(* IEC 61131-3 sources: AXOpen/src/components.dukane.welders/ctrl/src/TemplateComponent (part 2) *)

                IF Config.HWIDs.HwID_out_1  = UINT#0 THEN
                    Messenger.Activate(UINT#1152,eAxoMessageCategory#Error);
                    Status.Error.Id := UINT#1152;
                    RETURN;
                END_IF;
                IF Config.HWIDs.HwID_out_2  = UINT#0 THEN
                    Messenger.Activate(UINT#1153,eAxoMessageCategory#Error);
                    Status.Error.Id := UINT#1153;
                    RETURN;
                END_IF;
                IF Config.HWIDs.HwID_out_3  = UINT#0 THEN
                    Messenger.Activate(UINT#1154,eAxoMessageCategory#Error);
                    Status.Error.Id := UINT#1154;
                    RETURN;
                END_IF;
                IF Config.HWIDs.HwID_out_4  = UINT#0 THEN
                    Messenger.Activate(UINT#1155,eAxoMessageCategory#Error);
                    Status.Error.Id := UINT#1155;
                    RETURN;
                END_IF;
                IF Config.HWIDs.HwID_out_5  = UINT#0 THEN
                    Messenger.Activate(UINT#1156,eAxoMessageCategory#Error);
                    Status.Error.Id := UINT#1156;
                    RETURN;
                END_IF;
                IF Config.HWIDs.HwID_out_6  = UINT#0 THEN
                    Messenger.Activate(UINT#1157,eAxoMessageCategory#Error);
                    Status.Error.Id := UINT#1157;
                    RETURN;
                END_IF;
                IF Config.HWIDs.HwID_out_7  = UINT#0 THEN
                    Messenger.Activate(UINT#1158,eAxoMessageCategory#Error);
                    Status.Error.Id := UINT#1158;
                    RETURN;
                END_IF;
                IF Config.HWIDs.HwID_out_8  = UINT#0 THEN
                    Messenger.Activate(UINT#1159,eAxoMessageCategory#Error);
                    Status.Error.Id := UINT#1159;
                    RETURN;
                END_IF;
                IF Config.HWIDs.HwID_out_9  = UINT#0 THEN
                    Messenger.Activate(UINT#1160,eAxoMessageCategory#Error);
                    Status.Error.Id := UINT#1160;
                    RETURN;
                END_IF;
                IF Config.HWIDs.HwID_out_10  = UINT#0 THEN
                    Messenger.Activate(UINT#1161,eAxoMessageCategory#Error);
                    Status.Error.Id := UINT#1161;
                    RETURN;
                END_IF;
                IF Config.HWIDs.HwID_out_11  = UINT#0 THEN
                    Messenger.Activate(UINT#1162,eAxoMessageCategory#Error);
                    Status.Error.Id := UINT#1162;
                    RETURN;
                END_IF;
                IF Config.HWIDs.HwID_out_12  = UINT#0 THEN
                    Messenger.Activate(UINT#1163,eAxoMessageCategory#Error);
                    Status.Error.Id := UINT#1163;
                    RETURN;
                END_IF;
                IF Config.HWIDs.HwID_out_13  = UINT#0 THEN
                    Messenger.Activate(UINT#1164,eAxoMessageCategory#Error);
                    Status.Error.Id := UINT#1164;
                    RETURN;
                END_IF;
                IF Config.HWIDs.HwID_out_14  = UINT#0 THEN
                    Messenger.Activate(UINT#1165,eAxoMessageCategory#Error);
                    Status.Error.Id := UINT#1165;
                    RETURN;
                END_IF;
                IF Config.HWIDs.HwID_out_15  = UINT#0 THEN
                    Messenger.Activate(UINT#1166,eAxoMessageCategory#Error);
                    Status.Error.Id := UINT#1166;
                    RETURN;
                END_IF;
                IF Config.HWIDs.HwID_out_16  = UINT#0 THEN
                    Messenger.Activate(UINT#1167,eAxoMessageCategory#Error);
                    Status.Error.Id := UINT#1167;
                    RETURN;
                END_IF;
                IF Config.HWIDs.HwID_out_17  = UINT#0 THEN
                    Messenger.Activate(UINT#1168,eAxoMessageCategory#Error);
                    Status.Error.Id := UINT#1168;
                    RETURN;
                END_IF;
                IF Config.HWIDs.HwID_out_18  = UINT#0 THEN
                    Messenger.Activate(UINT#1169,eAxoMessageCategory#Error);
                    Status.Error.Id := UINT#1169;
                    RETURN;
                END_IF;
                IF Config.HWIDs.HwID_out_19  = UINT#0 THEN
                    Messenger.Activate(UINT#1170,eAxoMessageCategory#Error);
                    Status.Error.Id := UINT#1170;
                    RETURN;
                END_IF;
                IF Config.HWIDs.HwID_out_20  = UINT#0 THEN
                    Messenger.Activate(UINT#1171,eAxoMessageCategory#Error);
                    Status.Error.Id := UINT#1171;
                    RETURN;
                END_IF;

                _initHwCheckDone    := TRUE;
            END_IF;

            //***********Update inputs **************
            _retVal := Siemens.Simatic.S71500.DistributedIO.ReadData(TO_WORD(Config.HWIDs.HwID_in_1) ,_data_in);
            IF _retVal > WORD#0 THEN
                Messenger.Activate(UINT#1201, eAxoMessageCategory#ProgrammingError);
                Status.Error.Id := UINT#1201;
                RETURN;
            END_IF;

            // TemplateComponentInputStructure_hwID_in_1.Item1  :=      _data_in[0].%X0;
            // TemplateComponentInputStructure_hwID_in_1.Item2  :=      _data_in[0].%X1;
            // TemplateComponentInputStructure_hwID_in_1.Item3  :=      _data_in[0].%X2;
            // TemplateComponentInputStructure_hwID_in_1.Item4  :=      _data_in[0].%X3;
            // TemplateComponentInputStructure_hwID_in_1.Item5  :=      _data_in[0].%X4;

            _retVal := Siemens.Simatic.S71500.DistributedIO.ReadData(TO_WORD(Config.HWIDs.HwID_in_2) ,_data_in);
            IF _retVal > WORD#0 THEN
                Messenger.Activate(UINT#1202, eAxoMessageCategory#ProgrammingError);
                Status.Error.Id := UINT#1202;
                RETURN;
            END_IF;

            // TemplateComponentInputStructure_hwID_in_2.Item1  :=      _data_in[0].%X0;
            // TemplateComponentInputStructure_hwID_in_2.Item2  :=      _data_in[0].%X1;
            // TemplateComponentInputStructure_hwID_in_2.Item3  :=      _data_in[0].%X2;
            // TemplateComponentInputStructure_hwID_in_2.Item4  :=      _data_in[0].%X3;
            // TemplateComponentInputStructure_hwID_in_2.Item5  :=      _data_in[0].%X4;

            _retVal := Siemens.Simatic.S71500.DistributedIO.ReadData(TO_WORD(Config.HWIDs.HwID_in_3) ,_data_in);
            IF _retVal > WORD#0 THEN
                Messenger.Activate(UINT#1203, eAxoMessageCategory#ProgrammingError);
                Status.Error.Id := UINT#1203;
                RETURN;
            END_IF;

            // TemplateComponentInputStructure_hwID_in_3.Item1  :=      _data_in[0].%X0;
            // TemplateComponentInputStructure_hwID_in_3.Item2  :=      _data_in[0].%X1;
            // TemplateComponentInputStructure_hwID_in_3.Item3  :=      _data_in[0].%X2;
            // TemplateComponentInputStructure_hwID_in_3.Item4  :=      _data_in[0].%X3;
            // TemplateComponentInputStructure_hwID_in_3.Item5  :=      _data_in[0].%X4;

            _retVal := Siemens.Simatic.S71500.DistributedIO.ReadData(TO_WORD(Config.HWIDs.HwID_in_4) ,_data_in);
            IF _retVal > WORD#0 THEN
                Messenger.Activate(UINT#1204, eAxoMessageCategory#ProgrammingError);
                Status.Error.Id := UINT#1204;
                RETURN;
            END_IF;

            // TemplateComponentInputStructure_hwID_in_4.Item1  :=      _data_in[0].%X0;
            // TemplateComponentInputStructure_hwID_in_4.Item2  :=      _data_in[0].%X1;
            // TemplateComponentInputStructure_hwID_in_4.Item3  :=      _data_in[0].%X2;
            // TemplateComponentInputStructure_hwID_in_4.Item4  :=      _data_in[0].%X3;
            // TemplateComponentInputStructure_hwID_in_4.Item5  :=      _data_in[0].%X4;

            _retVal := Siemens.Simatic.S71500.DistributedIO.ReadData(TO_WORD(Config.HWIDs.HwID_in_5) ,_data_in);
            IF _retVal > WORD#0 THEN
                Messenger.Activate(UINT#1205, eAxoMessageCategory#ProgrammingError);
                Status.Error.Id := UINT#1205;
                RETURN;
            END_IF;

            // TemplateComponentInputStructure_hwID_in_5.Item1  :=      _data_in[0].%X0;
            // TemplateComponentInputStructure_hwID_in_5.Item2  :=      _data_in[0].%X1;
            // TemplateComponentInputStructure_hwID_in_5.Item3  :=      _data_in[0].%X2;
            // TemplateComponentInputStructure_hwID_in_5.Item4  :=      _data_in[0].%X3;
            // TemplateComponentInputStructure_hwID_in_5.Item5  :=      _data_in[0].%X4;

            _retVal := Siemens.Simatic.S71500.DistributedIO.ReadData(TO_WORD(Config.HWIDs.HwID_in_6) ,_data_in);
            IF _retVal > WORD#0 THEN
                Messenger.Activate(UINT#1206, eAxoMessageCategory#ProgrammingError);
                Status.Error.Id := UINT#1206;
                RETURN;
            END_IF;

            // _word.%B1                                                           :=  _data_in[0];
            // _word.%B0                                                           :=  _data_in[1];
            // TemplateComponentInputStructure_hwID_in_6.Item1                     :=  TO_UINT(_word);
            // _word.%B1                                                           :=  _data_in[2];
            // _word.%B0                                                           :=  _data_in[3];
            // TemplateComponentInputStructure_hwID_in_6.Item2                     :=  TO_UINT(_word);
            // _word.%B1                                                           :=  _data_in[4];
            // _word.%B0                                                           :=  _data_in[5];
            // TemplateComponentInputStructure_hwID_in_6.Item3                     :=  TO_UINT(_word);
            // _word.%B1                                                           :=  _data_in[6];
            // _word.%B0                                                           :=  _data_in[7];
            // TemplateComponentInputStructure_hwID_in_6.Item4                     :=  TO_UINT(_word);

            _retVal := Siemens.Simatic.S71500.DistributedIO.ReadData(TO_WORD(Config.HWIDs.HwID_in_7) ,_data_in);
            IF _retVal > WORD#0 THEN
                Messenger.Activate(UINT#1207, eAxoMessageCategory#ProgrammingError);
                Status.Error.Id := UINT#1207;
                RETURN;
            END_IF;

            // _dword.%B3                                                          :=  _data_in[0];
            // _dword.%B2                                                          :=  _data_in[1];
            // _dword.%B1                                                          :=  _data_in[2];
            // _dword.%B0                                                          :=  _data_in[3];
            // TemplateComponentInputStructure_hwID_in_7.Item1                     :=  TO_DINT(_dword);
            // _dword.%B3                                                          :=  _data_in[4];
            // _dword.%B2                                                          :=  _data_in[5];
            // _dword.%B1                                                          :=  _data_in[6];
            // _dword.%B0                                                          :=  _data_in[7];
            // TemplateComponentInputStructure_hwID_in_7.Item2                     :=  TO_REAL(_dword);

            _retVal := Siemens.Simatic.S71500.DistributedIO.ReadData(TO_WORD(Config.HWIDs.HwID_in_8) ,_data_in);
            IF _retVal > WORD#0 THEN
                Messenger.Activate(UINT#1208, eAxoMessageCategory#ProgrammingError);
                Status.Error.Id := UINT#1208;
                RETURN;
            END_IF;

            // _dword.%B3                                                          :=  _data_in[0];
            // _dword.%B2                                                          :=  _data_in[1];
            // _dword.%B1                                                          :=  _data_in[2];
            // _dword.%B0                                                          :=  _data_in[3];
            // TemplateComponentInputStructure_hwID_in_8.Item1                     :=  TO_DINT(_dword);
            // _dword.%B3                                                          :=  _data_in[4];
            // _dword.%B2                                                          :=  _data_in[5];
            // _dword.%B1                                                          :=  _data_in[6];
            // _dword.%B0                                                          :=  _data_in[7];
            // TemplateComponentInputStructure_hwID_in_8.Item2                     :=  TO_REAL(_dword);

            _retVal := Siemens.Simatic.S71500.DistributedIO.ReadData(TO_WORD(Config.HWIDs.HwID_in_9) ,_data_in);
            IF _retVal > WORD#0 THEN
                Messenger.Activate(UINT#1209, eAxoMessageCategory#ProgrammingError);
                Status.Error.Id := UINT#1209;
                RETURN;
            END_IF;

            // _dword.%B3                                                          :=  _data_in[0];
            // _dword.%B2                                                          :=  _data_in[1];
            // _dword.%B1                                                          :=  _data_in[2];
            // _dword.%B0                                                          :=  _data_in[3];
            // TemplateComponentInputStructure_hwID_in_9.Item1                     :=  TO_DINT(_dword);
            // _dword.%B3                                                          :=  _data_in[4];
            // _dword.%B2                                                          :=  _data_in[5];
            // _dword.%B1                                                          :=  _data_in[6];
            // _dword.%B0                                                          :=  _data_in[7];
            // TemplateComponentInputStructure_hwID_in_9.Item2                     :=  TO_REAL(_dword);

            _retVal := Siemens.Simatic.S71500.DistributedIO.ReadData(TO_WORD(Config.HWIDs.HwID_in_10) ,_data_in);
            IF _retVal > WORD#0 THEN
                Messenger.Activate(UINT#1210, eAxoMessageCategory#ProgrammingError);
                Status.Error.Id := UINT#1210;
                RETURN;
            END_IF;

            // _dword.%B3                                                          :=  _data_in[0];
            // _dword.%B2                                                          :=  _data_in[1];
            // _dword.%B1                                                          :=  _data_in[2];
            // _dword.%B0                                                          :=  _data_in[3];
            // TemplateComponentInputStructure_hwID_in_10.Item1                    :=  TO_DINT(_dword);
            // _dword.%B3                                                          :=  _data_in[4];
            // _dword.%B2                                                          :=  _data_in[5];
            // _dword.%B1                                                          :=  _data_in[6];
            // _dword.%B0                                                          :=  _data_in[7];
            // TemplateComponentInputStructure_hwID_in_10.Item2                    :=  TO_REAL(_dword);

            _retVal := Siemens.Simatic.S71500.DistributedIO.ReadData(TO_WORD(Config.HWIDs.HwID_in_11) ,_data_in);
            IF _retVal > WORD#0 THEN
                Messenger.Activate(UINT#1211, eAxoMessageCategory#ProgrammingError);
                Status.Error.Id := UINT#1211;
                RETURN;
            END_IF;

            // TemplateComponentInputStructure_hwID_in_11.Item1  :=      _data_in[0].%X0;
            // TemplateComponentInputStructure_hwID_in_11.Item2  :=      _data_in[0].%X1;
            // TemplateComponentInputStructure_hwID_in_11.Item3  :=      _data_in[0].%X2;
            // TemplateComponentInputStructure_hwID_in_11.Item4  :=      _data_in[0].%X3;
            // TemplateComponentInputStructure_hwID_in_11.Item5  :=      _data_in[0].%X4;

            _retVal := Siemens.Simatic.S71500.DistributedIO.ReadData(TO_WORD(Config.HWIDs.HwID_in_12) ,_data_in);
            IF _retVal > WORD#0 THEN
                Messenger.Activate(UINT#1212, eAxoMessageCategory#ProgrammingError);
                Status.Error.Id := UINT#1212;
                RETURN;
            END_IF;

            // TemplateComponentInputStructure_hwID_in_12.Item1  :=      _data_in[0].%X0;
            // TemplateComponentInputStructure_hwID_in_12.Item2  :=      _data_in[0].%X1;
            // TemplateComponentInputStructure_hwID_in_12.Item3  :=      _data_in[0].%X2;
            // TemplateComponentInputStructure_hwID_in_12.Item4  :=      _data_in[0].%X3;
            // TemplateComponentInputStructure_hwID_in_12.Item5  :=      _data_in[0].%X4;

            _retVal := Siemens.Simatic.S71500.DistributedIO.ReadData(TO_WORD(Config.HWIDs.HwID_in_13) ,_data_in);
            IF _retVal > WORD#0 THEN
                Messenger.Activate(UINT#1213, eAxoMessageCategory#ProgrammingError);
                Status.Error.Id := UINT#1213;
                RETURN;
            END_IF;

            // TemplateComponentInputStructure_hwID_in_13.Item1  :=      _data_in[0].%X0;
            // TemplateComponentInputStructure_hwID_in_13.Item2  :=      _data_in[0].%X1;
            // TemplateComponentInputStructure_hwID_in_13.Item3  :=      _data_in[0].%X2;
            // TemplateComponentInputStructure_hwID_in_13.Item4  :=      _data_in[0].%X3;
            // TemplateComponentInputStructure_hwID_in_13.Item5  :=      _data_in[0].%X4;

            _retVal := Siemens.Simatic.S71500.DistributedIO.ReadData(TO_WORD(Config.HWIDs.HwID_in_14) ,_data_in);
            IF _retVal > WORD#0 THEN
                Messenger.Activate(UINT#1214, eAxoMessageCategory#ProgrammingError);
                Status.Error.Id := UINT#1214;
                RETURN;
            END_IF;

            // TemplateComponentInputStructure_hwID_in_14.Item1  :=      _data_in[0].%X0;
            // TemplateComponentInputStructure_hwID_in_14.Item2  :=      _data_in[0].%X1;
            // TemplateComponentInputStructure_hwID_in_14.Item3  :=      _data_in[0].%X2;
            // TemplateComponentInputStructure_hwID_in_14.Item4  :=      _data_in[0].%X3;
            // TemplateComponentInputStructure_hwID_in_14.Item5  :=      _data_in[0].%X4;

            _retVal := Siemens.Simatic.S71500.DistributedIO.ReadData(TO_WORD(Config.HWIDs.HwID_in_15) ,_data_in);
            IF _retVal > WORD#0 THEN
                Messenger.Activate(UINT#1215, eAxoMessageCategory#ProgrammingError);
                Status.Error.Id := UINT#1215;
                RETURN;
            END_IF;

            // TemplateComponentInputStructure_hwID_in_15.Item1  :=      _data_in[0].%X0;
            // TemplateComponentInputStructure_hwID_in_15.Item2  :=      _data_in[0].%X1;
            // TemplateComponentInputStructure_hwID_in_15.Item3  :=      _data_in[0].%X2;
            // TemplateComponentInputStructure_hwID_in_15.Item4  :=      _data_in[0].%X3;
            // TemplateComponentInputStructure_hwID_in_15.Item5  :=      _data_in[0].%X4;

            _retVal := Siemens.Simatic.S71500.DistributedIO.ReadData(TO_WORD(Config.HWIDs.HwID_in_16) ,_data_in);
            IF _retVal > WORD#0 THEN
                Messenger.Activate(UINT#1216, eAxoMessageCategory#ProgrammingError);
                Status.Error.Id := UINT#1216;
                RETURN;
            END_IF;

            // _word.%B1                                                           :=  _data_in[0];
            // _word.%B0                                                           :=  _data_in[1];
            // TemplateComponentInputStructure_hwID_in_16.Item1                    :=  TO_UINT(_word);
            // _word.%B1                                                           :=  _data_in[2];
            // _word.%B0                                                           :=  _data_in[3];
            // TemplateComponentInputStructure_hwID_in_16.Item2                    :=  TO_UINT(_word);
            // _word.%B1                                                           :=  _data_in[4];
            // _word.%B0                                                           :=  _data_in[5];
            // TemplateComponentInputStructure_hwID_in_16.Item3                    :=  TO_UINT(_word);
            // _word.%B1                                                           :=  _data_in[6];
            // _word.%B0                                                           :=  _data_in[7];
            // TemplateComponentInputStructure_hwID_in_16.Item4                    :=  TO_UINT(_word);

            _retVal := Siemens.Simatic.S71500.DistributedIO.ReadData(TO_WORD(Config.HWIDs.HwID_in_17) ,_data_in);
            IF _retVal > WORD#0 THEN
                Messenger.Activate(UINT#1217, eAxoMessageCategory#ProgrammingError);
                Status.Error.Id := UINT#1217;
                RETURN;
            END_IF;

            // _dword.%B3                                                          :=  _data_in[0];
            // _dword.%B2                                                          :=  _data_in[1];
            // _dword.%B1                                                          :=  _data_in[2];
            // _dword.%B0                                                          :=  _data_in[3];
            // TemplateComponentInputStructure_hwID_in_17.Item1                    :=  TO_DINT(_dword);
            // _dword.%B3                                                          :=  _data_in[4];
            // _dword.%B2                                                          :=  _data_in[5];
            // _dword.%B1                                                          :=  _data_in[6];
            // _dword.%B0                                                          :=  _data_in[7];
            // TemplateComponentInputStructure_hwID_in_17.Item2                    :=  TO_REAL(_dword);

            _retVal := Siemens.Simatic.S71500.DistributedIO.ReadData(TO_WORD(Config.HWIDs.HwID_in_18) ,_data_in);
            IF _retVal > WORD#0 THEN
                Messenger.Activate(UINT#1218, eAxoMessageCategory#ProgrammingError);
                Status.Error.Id := UINT#1218;
                RETURN;
            END_IF;

            // _dword.%B3                                                          :=  _data_in[0];
            // _dword.%B2                                                          :=  _data_in[1];
            // _dword.%B1                                                          :=  _data_in[2];
            // _dword.%B0                                                          :=  _data_in[3];
            // TemplateComponentInputStructure_hwID_in_18.Item1                    :=  TO_DINT(_dword);
            // _dword.%B3                                                          :=  _data_in[4];
            // _dword.%B2                                                          :=  _data_in[5];
            // _dword.%B1                                                          :=  _data_in[6];
            // _dword.%B0                                                          :=  _data_in[7];
            // TemplateComponentInputStructure_hwID_in_18.Item2                    :=  TO_REAL(_dword);

            _retVal := Siemens.Simatic.S71500.DistributedIO.ReadData(TO_WORD(Config.HWIDs.HwID_in_19) ,_data_in);
            IF _retVal > WORD#0 THEN
                Messenger.Activate(UINT#1219, eAxoMessageCategory#ProgrammingError);
                Status.Error.Id := UINT#1219;
                RETURN;
            END_IF;

            // _dword.%B3                                                          :=  _data_in[0];
            // _dword.%B2                                                          :=  _data_in[1];
            // _dword.%B1                                                          :=  _data_in[2];
            // _dword.%B0                                                          :=  _data_in[3];
            // TemplateComponentInputStructure_hwID_in_19.Item1                    :=  TO_DINT(_dword);
            // _dword.%B3                                                          :=  _data_in[4];
            // _dword.%B2                                                          :=  _data_in[5];
            // _dword.%B1                                                          :=  _data_in[6];
            // _dword.%B0                                                          :=  _data_in[7];
            // TemplateComponentInputStructure_hwID_in_19.Item2                    :=  TO_REAL(_dword);

            _retVal := Siemens.Simatic.S71500.DistributedIO.ReadData(TO_WORD(Config.HWIDs.HwID_in_20) ,_data_in);
            IF _retVal > WORD#0 THEN
                Messenger.Activate(UINT#1220, eAxoMessageCategory#ProgrammingError);
                Status.Error.Id := UINT#1220;
                RETURN;
            END_IF;

            // _dword.%B3                                                          :=  _data_in[0];
            // _dword.%B2                                                          :=  _data_in[1];
            // _dword.%B1                                                          :=  _data_in[2];
            // _dword.%B0                                                          :=  _data_in[3];
            // TemplateComponentInputStructure_hwID_in_20.Item1                    :=  TO_DINT(_dword);
            // _dword.%B3                                                          :=  _data_in[4];
            // _dword.%B2                                                          :=  _data_in[5];
            // _dword.%B1                                                          :=  _data_in[6];
            // _dword.%B0                                                          :=  _data_in[7];
            // TemplateComponentInputStructure_hwID_in_20.Item2                    :=  TO_REAL(_dword);

            //*************INITIALIZATION*************
            RestoreTask.Run(THIS);
            TemplateTask_10steps_1.Run(THIS);
            TemplateTask_10steps_2.Run(THIS);
            TemplateTask_10steps_3.Run(THIS);
            TemplateTask_10steps_4.Run(THIS);
            TemplateTask_10steps_5.Run(THIS);
            TemplateTask_10steps_6.Run(THIS);
            TemplateTask_20steps_1.Run(THIS);
            TemplateTask_20steps_2.Run(THIS);
            TemplateTask_20steps_3.Run(THIS);
            TemplateTask_20steps_4.Run(THIS);
            TemplateTask_20steps_5.Run(THIS);
            TemplateTask_20steps_6.Run(THIS);

            //****************************************

            //********************Diagnostics*********
            HardwareDiagnosticsTask.Run(THIS,Config.HWIDs.HW_Device);
            //****************************************

            //*************RESTORE********************
            RestoreTask.SetIsDisabled(FALSE);
            IF RestoreTask.Execute(THIS) THEN
                THIS.Restore();
            END_IF;
            //****************************************

            //*************TemplateTask_10steps_1**************
            TemplateTask_10steps_1.SetIsDisabled(FALSE);
            IF TemplateTask_10steps_1.StartTriggered() THEN
                Status.Action.Id :=  UINT#100;
            END_IF;
            Messenger.ActivateOnCondition(ULINT#100,TemplateTask_10steps_1.IsBusy(), eAxoMessageCategory#Info);
            Messenger.ActivateOnCondition(ULINT#101,TemplateTask_10steps_1.IsDone(), eAxoMessageCategory#Info);
            IF TemplateTask_10steps_1.Execute(THIS) THEN
                IF _progress = 0 THEN
                    Status.Error.Id := UINT#0;
                    TaskMessenger.Restore();
                    THIS.CallTimers(FALSE);
                    _progress := 300;
                END_IF;

                IF _progress = 300 THEN                                                                                     // TemplateTask_10steps_1 running: , add_the_detailed_description_of_the_current_action_1
                    IF _infoTimer.output THEN
                        TaskMessenger.Activate( UINT#500, eAxoMessageCategory#Warning);
                        Status.Error.Id :=      UINT#500;
                    END_IF;

                    IF TRUE THEN
                        THIS.CallTimers(FALSE);
                        _progress := 301;
                    END_IF;
                END_IF;

                IF _progress = 301 THEN                                                                                     // TemplateTask_10steps_1 running: , add_the_detailed_description_of_the_current_action_2
                    IF _infoTimer.output THEN
                        TaskMessenger.Activate( UINT#501, eAxoMessageCategory#Warning);
                        Status.Error.Id :=      UINT#501;
                    END_IF;

                    IF TRUE THEN
                        THIS.CallTimers(FALSE);
                        _progress := 302;
                    END_IF;
                END_IF;

                IF _progress = 302 THEN                                                                                     // TemplateTask_10steps_1 running: , add_the_detailed_description_of_the_current_action_3
                    IF _infoTimer.output THEN
                        TaskMessenger.Activate( UINT#502, eAxoMessageCategory#Warning);
                        Status.Error.Id :=      UINT#502;
                    END_IF;

                    IF TRUE THEN
                        THIS.CallTimers(FALSE);
                        _progress := 303;
                    END_IF;
                END_IF;

                IF _progress = 303 THEN                                                                                     // TemplateTask_10steps_1 running: , add_the_detailed_description_of_the_current_action_4
                    IF _infoTimer.output THEN
                        TaskMessenger.Activate( UINT#503, eAxoMessageCategory#Warning);
                        Status.Error.Id :=      UINT#503;
                    END_IF;

                    IF TRUE THEN
                        THIS.CallTimers(FALSE);
                        _progress := 304;
                    END_IF;
                END_IF;

                IF _progress = 304 THEN                                                                                     // TemplateTask_10steps_1 running: , add_the_detailed_description_of_the_current_action_5
                    IF _infoTimer.output THEN
                        TaskMessenger.Activate( UINT#504, eAxoMessageCategory#Warning);
                        Status.Error.Id :=      UINT#504;
                    END_IF;

                    IF TRUE THEN
                        THIS.CallTimers(FALSE);
                        _progress := 305;
                    END_IF;
                END_IF;

                IF _progress = 305 THEN                                                                                     // TemplateTask_10steps_1 running: , add_the_detailed_description_of_the_current_action_6
                    IF _infoTimer.output THEN
                        TaskMessenger.Activate( UINT#505, eAxoMessageCategory#Warning);
                        Status.Error.Id :=      UINT#505;
                    END_IF;

                    IF TRUE THEN
                        THIS.CallTimers(FALSE);
                        _progress := 306;
                    END_IF;
                END_IF;

                IF _progress = 306 THEN                                                                                     // TemplateTask_10steps_1 running: , add_the_detailed_description_of_the_current_action_7
                    IF _infoTimer.output THEN
                        TaskMessenger.Activate( UINT#506, eAxoMessageCategory#Warning);
                        Status.Error.Id :=      UINT#506;
                    END_IF;

                    IF TRUE THEN
                        THIS.CallTimers(FALSE);
                        _progress := 307;
                    END_IF;
                END_IF;

                IF _progress = 307 THEN                                                                                     // TemplateTask_10steps_1 running: , add_the_detailed_description_of_the_current_action_8
                    IF _infoTimer.output THEN
                        TaskMessenger.Activate( UINT#507, eAxoMessageCategory#Warning);
                        Status.Error.Id :=      UINT#507;
                    END_IF;

                    IF TRUE THEN
                        THIS.CallTimers(FALSE);
                        _progress := 308;
                    END_IF;
                END_IF;

                IF _progress = 308 THEN                                                                                     // TemplateTask_10steps_1 running: , add_the_detailed_description_of_the_current_action_9
                    IF _infoTimer.output THEN
                        TaskMessenger.Activate( UINT#508, eAxoMessageCategory#Warning);
                        Status.Error.Id :=      UINT#508;
                    END_IF;

                    IF TRUE THEN
                        THIS.CallTimers(FALSE);
                        _progress := 309;
                    END_IF;
                END_IF;

                IF _progress = 309 THEN                                                                                     // TemplateTask_10steps_1 running: , add_the_detailed_description_of_the_current_action_10
                    TemplateTask_10steps_1.DoneWhen(TRUE);
                    _progress := 0;
                END_IF;

                THIS.CallTimers(TRUE);

                TemplateTask_10steps_1.ThrowWhen(_errorTimer.output);
                Status.Action.Id := TO_UINT(_progress);
                TemplateTask_10steps_1.ThrowWhen(TemplateTask_10steps_1.Duration >= Config.TaskTimeout AND Config.TaskTimeout > T#0s ,'TemplateTask_10steps_1 timeout.');
            END_IF;
            IF TemplateTask_10steps_1.DoneReached() THEN
                Status.Action.Id :=  UINT#101;
                Status.Error.Id :=  UINT#0;
            ELSIF TemplateTask_10steps_1.ErrorOccured() THEN
                Status.Action.Id :=  UINT#10000;
                Status.Error.Id  :=  UINT#10000;
            ELSIF TemplateTask_10steps_1.AbortTriggered()THEN
                Status.Action.Id :=  UINT#10001;
                Status.Error.Id  :=  UINT#10001;
            END_IF;
            Messenger.ActivateOnCondition(ULINT#10000,TemplateTask_10steps_1.HasError(), eAxoMessageCategory#Error);
            Messenger.ActivateOnCondition(ULINT#10001,TemplateTask_10steps_1.IsAborted(), eAxoMessageCategory#Error);
            Messenger.ActivateOnCondition(ULINT#102,TemplateTask_10steps_1.RestoreTriggered() , eAxoMessageCategory#Error);
            IF TemplateTask_10steps_1.RestoreTriggered() AND _progress >= 300 AND _progress <= 309  THEN
                Status.Action.Id :=  UINT#102;
                _progress := 0;
            END_IF;
            //**************************************************

            //*************TemplateTask_10steps_2***************
            TemplateTask_10steps_2.SetIsDisabled(FALSE);
            IF TemplateTask_10steps_2.StartTriggered() THEN
                Status.Action.Id :=  UINT#110;
            END_IF;
            Messenger.ActivateOnCondition(ULINT#110,TemplateTask_10steps_2.IsBusy(), eAxoMessageCategory#Info);
            Messenger.ActivateOnCondition(ULINT#111,TemplateTask_10steps_2.IsDone(), eAxoMessageCategory#Info);
            IF TemplateTask_10steps_2.Execute(THIS) THEN
                IF _progress = 0 THEN
                    Status.Error.Id := UINT#0;
                    TaskMessenger.Restore();
                    THIS.CallTimers(FALSE);
                    _progress := 310;
                END_IF;

                IF _progress = 310 THEN                                                                                     // TemplateTask_10steps_2 running: , add_the_detailed_description_of_the_current_action_1
                    IF _infoTimer.output THEN
                        TaskMessenger.Activate( UINT#510, eAxoMessageCategory#Warning);
                        Status.Error.Id :=      UINT#510;
                    END_IF;

                    IF TRUE THEN
                        THIS.CallTimers(FALSE);
                        _progress := 311;
                    END_IF;
                END_IF;

                IF _progress = 311 THEN                                                                                     // TemplateTask_10steps_2 running: , add_the_detailed_description_of_the_current_action_2
                    IF _infoTimer.output THEN
                        TaskMessenger.Activate( UINT#511, eAxoMessageCategory#Warning);
                        Status.Error.Id :=      UINT#511;
                    END_IF;

                    IF TRUE THEN
                        THIS.CallTimers(FALSE);
                        _progress := 312;
                    END_IF;
                END_IF;

                IF _progress = 312 THEN                                                                                     // TemplateTask_10steps_2 running: , add_the_detailed_description_of_the_current_action_3
                    IF _infoTimer.output THEN
                        TaskMessenger.Activate( UINT#512, eAxoMessageCategory#Warning);
                        Status.Error.Id :=      UINT#512;
                    END_IF;

                    IF TRUE THEN
                        THIS.CallTimers(FALSE);
                        _progress := 313;
                    END_IF;
                END_IF;

                IF _progress = 313 THEN                                                                                     // TemplateTask_10steps_2 running: , add_the_detailed_description_of_the_current_action_4
                    IF _infoTimer.output THEN
                        TaskMessenger.Activate( UINT#513, eAxoMessageCategory#Warning);
                        Status.Error.Id :=      UINT#513;
                    END_IF;

                    IF TRUE THEN
                        THIS.CallTimers(FALSE);
                        _progress := 314;
                    END_IF;
                END_IF;

                IF _progress = 314 THEN                                                                                     // TemplateTask_10steps_2 running: , add_the_detailed_description_of_the_current_action_5
                    IF _infoTimer.output THEN
                        TaskMessenger.Activate( UINT#514, eAxoMessageCategory#Warning);
                        Status.Error.Id :=      UINT#514;
                    END_IF;

                    IF TRUE THEN
                        THIS.CallTimers(FALSE);
                        _progress := 315;
                    END_IF;
                END_IF;

                IF _progress = 315 THEN                                                                                     // TemplateTask_10steps_2 running: , add_the_detailed_description_of_the_current_action_6
                    IF _infoTimer.output THEN
                        TaskMessenger.Activate( UINT#515, eAxoMessageCategory#Warning);
                        Status.Error.Id :=      UINT#515;
                    END_IF;

                    IF TRUE THEN
                        THIS.CallTimers(FALSE);
                        _progress := 316;
                    END_IF;
                END_IF;

                IF _progress = 316 THEN                                                                                     // TemplateTask_10steps_2 running: , add_the_detailed_description_of_the_current_action_7
                    IF _infoTimer.output THEN
                        TaskMessenger.Activate( UINT#516, eAxoMessageCategory#Warning);
                        Status.Error.Id :=      UINT#516;
                    END_IF;

                    IF TRUE THEN
                        THIS.CallTimers(FALSE);
                        _progress := 317;
                    END_IF;
                END_IF;

                IF _progress = 317 THEN                                                                                     // TemplateTask_10steps_2 running: , add_the_detailed_description_of_the_current_action_8
                    IF _infoTimer.output THEN
                        TaskMessenger.Activate( UINT#517, eAxoMessageCategory#Warning);
                        Status.Error.Id :=      UINT#517;
                    END_IF;

                    IF TRUE THEN
                        THIS.CallTimers(FALSE);
                        _progress := 318;
                    END_IF;
                END_IF;

                IF _progress = 318 THEN                                                                                     // TemplateTask_10steps_2 running: , add_the_detailed_description_of_the_current_action_9
                    IF _infoTimer.output THEN
                        TaskMessenger.Activate( UINT#518, eAxoMessageCategory#Warning);
                        Status.Error.Id :=      UINT#518;
                    END_IF;

                    IF TRUE THEN
                        THIS.CallTimers(FALSE);
                        _progress := 319;
                    END_IF;
                END_IF;

                IF _progress = 319 THEN                                                                                     // TemplateTask_10steps_2 running: , add_the_detailed_description_of_the_current_action_10
                    TemplateTask_10steps_2.DoneWhen(TRUE);
                    _progress := 0;
                END_IF;

                THIS.CallTimers(TRUE);

                TemplateTask_10steps_2.ThrowWhen(_errorTimer.output);
                Status.Action.Id := TO_UINT(_progress);
                TemplateTask_10steps_2.ThrowWhen(TemplateTask_10steps_2.Duration >= Config.TaskTimeout AND Config.TaskTimeout > T#0s ,'TemplateTask_10steps_2 timeout.');
            END_IF;
            IF TemplateTask_10steps_2.DoneReached() THEN
                Status.Action.Id :=  UINT#111;
                Status.Error.Id :=  UINT#0;
            ELSIF TemplateTask_10steps_2.ErrorOccured() THEN
                Status.Action.Id :=  UINT#10010;
                Status.Error.Id  :=  UINT#10010;
            ELSIF TemplateTask_10steps_2.AbortTriggered()THEN
                Status.Action.Id :=  UINT#10011;
                Status.Error.Id  :=  UINT#10011;
            END_IF;
            Messenger.ActivateOnCondition(ULINT#10010,TemplateTask_10steps_2.HasError(), eAxoMessageCategory#Error);
            Messenger.ActivateOnCondition(ULINT#10011,TemplateTask_10steps_2.IsAborted(), eAxoMessageCategory#Error);
            Messenger.ActivateOnCondition(ULINT#112,TemplateTask_10steps_2.RestoreTriggered() , eAxoMessageCategory#Error);
            IF TemplateTask_10steps_2.RestoreTriggered() AND _progress >= 310 AND _progress <= 319  THEN
                Status.Action.Id :=  UINT#112;
                _progress := 0;
            END_IF;
            //**************************************************

            //*************TemplateTask_10steps_3***************
            TemplateTask_10steps_3.SetIsDisabled(FALSE);
            IF TemplateTask_10steps_3.StartTriggered() THEN
                Status.Action.Id :=  UINT#120;
            END_IF;
            Messenger.ActivateOnCondition(ULINT#120,TemplateTask_10steps_3.IsBusy(), eAxoMessageCategory#Info);
            Messenger.ActivateOnCondition(ULINT#121,TemplateTask_10steps_3.IsDone(), eAxoMessageCategory#Info);
            IF TemplateTask_10steps_3.Execute(THIS) THEN
                IF _progress = 0 THEN
                    Status.Error.Id := UINT#0;
                    TaskMessenger.Restore();
                    THIS.CallTimers(FALSE);
                    _progress := 320;
                END_IF;

                IF _progress = 320 THEN                                                                                     // TemplateTask_10steps_3 running: , add_the_detailed_description_of_the_current_action_1
                    IF _infoTimer.output THEN
                        TaskMessenger.Activate( UINT#520, eAxoMessageCategory#Warning);
                        Status.Error.Id :=      UINT#520;
                    END_IF;

                    IF TRUE THEN
                        THIS.CallTimers(FALSE);
                        _progress := 321;
                    END_IF;
                END_IF;

                IF _progress = 321 THEN                                                                                     // TemplateTask_10steps_3 running: , add_the_detailed_description_of_the_current_action_2
                    IF _infoTimer.output THEN
                        TaskMessenger.Activate( UINT#521, eAxoMessageCategory#Warning);
                        Status.Error.Id :=      UINT#521;
                    END_IF;

                    IF TRUE THEN
                        THIS.CallTimers(FALSE);
                        _progress := 322;
                    END_IF;
                END_IF;

                IF _progress = 322 THEN                                                                                     // TemplateTask_10steps_3 running: , add_the_detailed_description_of_the_current_action_3
                    IF _infoTimer.output THEN
                        TaskMessenger.Activate( UINT#522, eAxoMessageCategory#Warning);
                        Status.Error.Id :=      UINT#522;
                    END_IF;

                    IF TRUE THEN
                        THIS.CallTimers(FALSE);
                        _progress := 323;
                    END_IF;
                END_IF;

                IF _progress = 323 THEN                                                                                     // TemplateTask_10steps_3 running: , add_the_detailed_description_of_the_current_action_4
                    IF _infoTimer.output THEN
                        TaskMessenger.Activate( UINT#523, eAxoMessageCategory#Warning);
                        Status.Error.Id :=      UINT#523;
                    END_IF;

                    IF TRUE THEN
                        THIS.CallTimers(FALSE);
                        _progress := 324;
                    END_IF;
                END_IF;

                IF _progress = 324 THEN                                                                                     // TemplateTask_10steps_3 running: , add_the_detailed_description_of_the_current_action_5
                    IF _infoTimer.output THEN
                        TaskMessenger.Activate( UINT#524, eAxoMessageCategory#Warning);
                        Status.Error.Id :=      UINT#524;
                    END_IF;

                    IF TRUE THEN
                        THIS.CallTimers(FALSE);
                        _progress := 325;
                    END_IF;
                END_IF;

                IF _progress = 325 THEN                                                                                     // TemplateTask_10steps_3 running: , add_the_detailed_description_of_the_current_action_6
                    IF _infoTimer.output THEN
                        TaskMessenger.Activate( UINT#525, eAxoMessageCategory#Warning);
                        Status.Error.Id :=      UINT#525;
                    END_IF;

                    IF TRUE THEN
                        THIS.CallTimers(FALSE);
                        _progress := 326;
                    END_IF;
                END_IF;

                IF _progress = 326 THEN                                                                                     // TemplateTask_10steps_3 running: , add_the_detailed_description_of_the_current_action_7
                    IF _infoTimer.output THEN
                        TaskMessenger.Activate( UINT#526, eAxoMessageCategory#Warning);
                        Status.Error.Id :=      UINT#526;
                    END_IF;

                    IF TRUE THEN
                        THIS.CallTimers(FALSE);
                        _progress := 327;
                    END_IF;
                END_IF;

                IF _progress = 327 THEN                                                                                     // TemplateTask_10steps_3 running: , add_the_detailed_description_of_the_current_action_8
                    IF _infoTimer.output THEN
                        TaskMessenger.Activate( UINT#527, eAxoMessageCategory#Warning);
                        Status.Error.Id :=      UINT#527;
                    END_IF;

                    IF TRUE THEN
                        THIS.CallTimers(FALSE);
                        _progress := 328;
                    END_IF;
                END_IF;

                IF _progress = 328 THEN                                                                                     // TemplateTask_10steps_3 running: , add_the_detailed_description_of_the_current_action_9
                    IF _infoTimer.output THEN
                        TaskMessenger.Activate( UINT#528, eAxoMessageCategory#Warning);
                        Status.Error.Id :=      UINT#528;
                    END_IF;

                    IF TRUE THEN
                        THIS.CallTimers(FALSE);
                        _progress := 329;
                    END_IF;
                END_IF;

                IF _progress = 329 THEN                                                                                     // TemplateTask_10steps_3 running: , add_the_detailed_description_of_the_current_action_10
                    TemplateTask_10steps_3.DoneWhen(TRUE);
                    _progress := 0;
                END_IF;

                THIS.CallTimers(TRUE);

                TemplateTask_10steps_3.ThrowWhen(_errorTimer.output);
                Status.Action.Id := TO_UINT(_progress);
                TemplateTask_10steps_3.ThrowWhen(TemplateTask_10steps_3.Duration >= Config.TaskTimeout AND Config.TaskTimeout > T#0s ,'TemplateTask_10steps_3 timeout.');
            END_IF;
            IF TemplateTask_10steps_3.DoneReached() THEN
                Status.Action.Id :=  UINT#121;
                Status.Error.Id :=  UINT#0;
            ELSIF TemplateTask_10steps_3.ErrorOccured() THEN
                Status.Action.Id :=  UINT#10020;
                Status.Error.Id  :=  UINT#10020;
            ELSIF TemplateTask_10steps_3.AbortTriggered()THEN
                Status.Action.Id :=  UINT#10021;
                Status.Error.Id  :=  UINT#10021;
            END_IF;
            Messenger.ActivateOnCondition(ULINT#10020,TemplateTask_10steps_3.HasError(), eAxoMessageCategory#Error);
            Messenger.ActivateOnCondition(ULINT#10021,TemplateTask_10steps_3.IsAborted(), eAxoMessageCategory#Error);
            Messenger.ActivateOnCondition(ULINT#122,TemplateTask_10steps_3.RestoreTriggered() , eAxoMessageCategory#Error);
            IF TemplateTask_10steps_3.RestoreTriggered() AND _progress >= 320 AND _progress <= 329  THEN
                Status.Action.Id :=  UINT#122;
                _progress := 0;
            END_IF;
            //**************************************************

            //*************TemplateTask_10steps_4***************
            TemplateTask_10steps_4.SetIsDisabled(FALSE);
            IF TemplateTask_10steps_4.StartTriggered() THEN
                Status.Action.Id :=  UINT#130;
            END_IF;
            Messenger.ActivateOnCondition(ULINT#130,TemplateTask_10steps_4.IsBusy(), eAxoMessageCategory#Info);
            Messenger.ActivateOnCondition(ULINT#131,TemplateTask_10steps_4.IsDone(), eAxoMessageCategory#Info);
            IF TemplateTask_10steps_4.Execute(THIS) THEN
                IF _progress = 0 THEN
                    Status.Error.Id := UINT#0;
                    TaskMessenger.Restore();
                    THIS.CallTimers(FALSE);
                    _progress := 330;
                END_IF;

                IF _progress = 330 THEN                                                                                     // TemplateTask_10steps_4 running: , add_the_detailed_description_of_the_current_action_1
                    IF _infoTimer.output THEN
                        TaskMessenger.Activate( UINT#530, eAxoMessageCategory#Warning);
                        Status.Error.Id :=      UINT#530;
                    END_IF;

                    IF TRUE THEN
                        THIS.CallTimers(FALSE);
                        _progress := 331;
                    END_IF;
                END_IF;

                IF _progress = 331 THEN                                                                                     // TemplateTask_10steps_4 running: , add_the_detailed_description_of_the_current_action_2
                    IF _infoTimer.output THEN
                        TaskMessenger.Activate( UINT#531, eAxoMessageCategory#Warning);
                        Status.Error.Id :=      UINT#531;
                    END_IF;

                    IF TRUE THEN
                        THIS.CallTimers(FALSE);
                        _progress := 332;
                    END_IF;
                END_IF;

                IF _progress = 332 THEN                                                                                     // TemplateTask_10steps_4 running: , add_the_detailed_description_of_the_current_action_3
                    IF _infoTimer.output THEN
                        TaskMessenger.Activate( UINT#532, eAxoMessageCategory#Warning);
                        Status.Error.Id :=      UINT#532;
                    END_IF;

                    IF TRUE THEN
                        THIS.CallTimers(FALSE);
                        _progress := 333;
                    END_IF;
                END_IF;

                IF _progress = 333 THEN                                                                                     // TemplateTask_10steps_4 running: , add_the_detailed_description_of_the_current_action_4
                    IF _infoTimer.output THEN
                        TaskMessenger.Activate( UINT#533, eAxoMessageCategory#Warning);
                        Status.Error.Id :=      UINT#533;
                    END_IF;

                    IF TRUE THEN
                        THIS.CallTimers(FALSE);
                        _progress := 334;
                    END_IF;
                END_IF;

                IF _progress = 334 THEN                                                                                     // TemplateTask_10steps_4 running: , add_the_detailed_description_of_the_current_action_5
                    IF _infoTimer.output THEN
                        TaskMessenger.Activate( UINT#534, eAxoMessageCategory#Warning);
                        Status.Error.Id :=      UINT#534;
                    END_IF;

                    IF TRUE THEN
                        THIS.CallTimers(FALSE);
                        _progress := 335;
                    END_IF;
                END_IF;

                IF _progress = 335 THEN                                                                                     // TemplateTask_10steps_4 running: , add_the_detailed_description_of_the_current_action_6
                    IF _infoTimer.output THEN
                        TaskMessenger.Activate( UINT#535, eAxoMessageCategory#Warning);
                        Status.Error.Id :=      UINT#535;
                    END_IF;

                    IF TRUE THEN
                        THIS.CallTimers(FALSE);
                        _progress := 336;
                    END_IF;
                END_IF;

                IF _progress = 336 THEN                                                                                     // TemplateTask_10steps_4 running: , add_the_detailed_description_of_the_current_action_7
                    IF _infoTimer.output THEN
                        TaskMessenger.Activate( UINT#536, eAxoMessageCategory#Warning);
                        Status.Error.Id :=      UINT#536;
                    END_IF;

                    IF TRUE THEN
                        THIS.CallTimers(FALSE);
                        _progress := 337;
                    END_IF;
                END_IF;

                IF _progress = 337 THEN                                                                                     // TemplateTask_10steps_4 running: , add_the_detailed_description_of_the_current_action_8
                    IF _infoTimer.output THEN
                        TaskMessenger.Activate( UINT#537, eAxoMessageCategory#Warning);
                        Status.Error.Id :=      UINT#537;
                    END_IF;

                    IF TRUE THEN
                        THIS.CallTimers(FALSE);
                        _progress := 338;
                    END_IF;
                END_IF;

                IF _progress = 338 THEN                                                                                     // TemplateTask_10steps_4 running: , add_the_detailed_description_of_the_current_action_9
                    IF _infoTimer.output THEN
                        TaskMessenger.Activate( UINT#538, eAxoMessageCategory#Warning);
                        Status.Error.Id :=      UINT#538;
                    END_IF;

                    IF TRUE THEN
                        THIS.CallTimers(FALSE);
                        _progress := 339;
                    END_IF;
                END_IF;

                IF _progress = 339 THEN                                                                                     // TemplateTask_10steps_4 running: , add_the_detailed_description_of_the_current_action_10
                    TemplateTask_10steps_4.DoneWhen(TRUE);
                    _progress := 0;
                END_IF;

                THIS.CallTimers(TRUE);

                TemplateTask_10steps_4.ThrowWhen(_errorTimer.output);
                Status.Action.Id := TO_UINT(_progress);
                TemplateTask_10steps_4.ThrowWhen(TemplateTask_10steps_4.Duration >= Config.TaskTimeout AND Config.TaskTimeout > T#0s ,'TemplateTask_10steps_4 timeout.');
            END_IF;
            IF TemplateTask_10steps_4.DoneReached() THEN
                Status.Action.Id :=  UINT#131;
                Status.Error.Id :=  UINT#0;
            ELSIF TemplateTask_10steps_4.ErrorOccured() THEN
                Status.Action.Id :=  UINT#10030;
                Status.Error.Id  :=  UINT#10030;
            ELSIF TemplateTask_10steps_4.AbortTriggered()THEN
                Status.Action.Id :=  UINT#10031;
                Status.Error.Id  :=  UINT#10031;
            END_IF;
            Messenger.ActivateOnCondition(ULINT#10030,TemplateTask_10steps_4.HasError(), eAxoMessageCategory#Error);
            Messenger.ActivateOnCondition(ULINT#10031,TemplateTask_10steps_4.IsAborted(), eAxoMessageCategory#Error);
            Messenger.ActivateOnCondition(ULINT#132,TemplateTask_10steps_4.RestoreTriggered() , eAxoMessageCategory#Error);
            IF TemplateTask_10steps_4.RestoreTriggered() AND _progress >= 330 AND _progress <= 339  THEN
                Status.Action.Id :=  UINT#132;
                _progress := 0;
            END_IF;
            //**************************************************

            //*************TemplateTask_10steps_5***************
            TemplateTask_10steps_5.SetIsDisabled(FALSE);
            IF TemplateTask_10steps_5.StartTriggered() THEN
                Status.Action.Id :=  UINT#140;
            END_IF;
            Messenger.ActivateOnCondition(ULINT#140,TemplateTask_10steps_5.IsBusy(), eAxoMessageCategory#Info);
            Messenger.ActivateOnCondition(ULINT#141,TemplateTask_10steps_5.IsDone(), eAxoMessageCategory#Info);
            IF TemplateTask_10steps_5.Execute(THIS) THEN
                IF _progress = 0 THEN
                    Status.Error.Id := UINT#0;
                    TaskMessenger.Restore();
                    THIS.CallTimers(FALSE);
                    _progress := 340;
                END_IF;

                IF _progress = 340 THEN                                                                                     // TemplateTask_10steps_5 running: , add_the_detailed_description_of_the_current_action_1
                    IF _infoTimer.output THEN
                        TaskMessenger.Activate( UINT#540, eAxoMessageCategory#Warning);
                        Status.Error.Id :=      UINT#540;
                    END_IF;

                    IF TRUE THEN
                        THIS.CallTimers(FALSE);
                        _progress := 341;
                    END_IF;
                END_IF;

                IF _progress = 341 THEN                                                                                     // TemplateTask_10steps_5 running: , add_the_detailed_description_of_the_current_action_2
                    IF _infoTimer.output THEN
                        TaskMessenger.Activate( UINT#541, eAxoMessageCategory#Warning);
                        Status.Error.Id :=      UINT#541;
                    END_IF;

                    IF TRUE THEN
                        THIS.CallTimers(FALSE);
                        _progress := 342;
                    END_IF;
                END_IF;

                IF _progress = 342 THEN                                                                                     // TemplateTask_10steps_5 running: , add_the_detailed_description_of_the_current_action_3
                    IF _infoTimer.output THEN
                        TaskMessenger.Activate( UINT#542, eAxoMessageCategory#Warning);
                        Status.Error.Id :=      UINT#542;
                    END_IF;

                    IF TRUE THEN
                        THIS.CallTimers(FALSE);
                        _progress := 343;
                    END_IF;
                END_IF;

                IF _progress = 343 THEN                                                                                     // TemplateTask_10steps_5 running: , add_the_detailed_description_of_the_current_action_4
                    IF _infoTimer.output THEN
                        TaskMessenger.Activate( UINT#543, eAxoMessageCategory#Warning);
                        Status.Error.Id :=      UINT#543;
                    END_IF;

                    IF TRUE THEN
                        THIS.CallTimers(FALSE);
                        _progress := 344;
                    END_IF;
                END_IF;

                IF _progress = 344 THEN                                                                                     // TemplateTask_10steps_5 running: , add_the_detailed_description_of_the_current_action_5
                    IF _infoTimer.output THEN
                        TaskMessenger.Activate( UINT#544, eAxoMessageCategory#Warning);
                        Status.Error.Id :=      UINT#544;
                    END_IF;

                    IF TRUE THEN
                        THIS.CallTimers(FALSE);
                        _progress := 345;
                    END_IF;
                END_IF;

                IF _progress = 345 THEN                                                                                     // TemplateTask_10steps_5 running: , add_the_detailed_description_of_the_current_action_6
                    IF _infoTimer.output THEN
                        TaskMessenger.Activate( UINT#545, eAxoMessageCategory#Warning);
                        Status.Error.Id :=      UINT#545;
                    END_IF;

                    IF TRUE THEN
                        THIS.CallTimers(FALSE);
                        _progress := 346;
                    END_IF;
                END_IF;

                IF _progress = 346 THEN                                                                                     // TemplateTask_10steps_5 running: , add_the_detailed_description_of_the_current_action_7
                    IF _infoTimer.output THEN
                        TaskMessenger.Activate( UINT#546, eAxoMessageCategory#Warning);
                        Status.Error.Id :=      UINT#546;
                    END_IF;

                    IF TRUE THEN
                        THIS.CallTimers(FALSE);
                        _progress := 347;
                    END_IF;
                END_IF;

                IF _progress = 347 THEN                                                                                     // TemplateTask_10steps_5 running: , add_the_detailed_description_of_the_current_action_8
                    IF _infoTimer.output THEN
                        TaskMessenger.Activate( UINT#547, eAxoMessageCategory#Warning);
                        Status.Error.Id :=      UINT#547;
                    END_IF;

                    IF TRUE THEN
                        THIS.CallTimers(FALSE);
                        _progress := 348;
                    END_IF;
                END_IF;

                IF _progress = 348 THEN                                                                                     // TemplateTask_10steps_5 running: , add_the_detailed_description_of_the_current_action_9
                    IF _infoTimer.output THEN
                        TaskMessenger.Activate( UINT#548, eAxoMessageCategory#Warning);
                        Status.Error.Id :=      UINT#548;
                    END_IF;

                    IF TRUE THEN
                        THIS.CallTimers(FALSE);
                        _progress := 349;
                    END_IF;
                END_IF;

                IF _progress = 349 THEN                                                                                     // TemplateTask_10steps_5 running: , add_the_detailed_description_of_the_current_action_10
                    TemplateTask_10steps_5.DoneWhen(TRUE);
                    _progress := 0;
                END_IF;

                THIS.CallTimers(TRUE);

                TemplateTask_10steps_5.ThrowWhen(_errorTimer.output);
                Status.Action.Id := TO_UINT(_progress);
                TemplateTask_10steps_5.ThrowWhen(TemplateTask_10steps_5.Duration >= Config.TaskTimeout AND Config.TaskTimeout > T#0s ,'TemplateTask_10steps_5 timeout.');
            END_IF;
            IF TemplateTask_10steps_5.DoneReached() THEN
                Status.Action.Id :=  UINT#141;
                Status.Error.Id :=  UINT#0;
            ELSIF TemplateTask_10steps_5.ErrorOccured() THEN
                Status.Action.Id :=  UINT#10040;
                Status.Error.Id  :=  UINT#10040;
            ELSIF TemplateTask_10steps_5.AbortTriggered()THEN
                Status.Action.Id :=  UINT#10041;
                Status.Error.Id  :=  UINT#10041;
            END_IF;
            Messenger.ActivateOnCondition(ULINT#10040,TemplateTask_10steps_5.HasError(), eAxoMessageCategory#Error);
            Messenger.ActivateOnCondition(ULINT#10041,TemplateTask_10steps_5.IsAborted(), eAxoMessageCategory#Error);
            Messenger.ActivateOnCondition(ULINT#142,TemplateTask_10steps_5.RestoreTriggered() , eAxoMessageCategory#Error);
            IF TemplateTask_10steps_5.RestoreTriggered() AND _progress >= 340 AND _progress <= 349  THEN
                Status.Action.Id :=  UINT#142;
                _progress := 0;
            END_IF;
            //**************************************************

            //*************TemplateTask_10steps_6***************
            TemplateTask_10steps_6.SetIsDisabled(FALSE);
            IF TemplateTask_10steps_6.StartTriggered() THEN
                Status.Action.Id :=  UINT#150;
            END_IF;
            Messenger.ActivateOnCondition(ULINT#150,TemplateTask_10steps_6.IsBusy(), eAxoMessageCategory#Info);
            Messenger.ActivateOnCondition(ULINT#151,TemplateTask_10steps_6.IsDone(), eAxoMessageCategory#Info);
            IF TemplateTask_10steps_6.Execute(THIS) THEN
                IF _progress = 0 THEN
                    Status.Error.Id := UINT#0;
                    TaskMessenger.Restore();
                    THIS.CallTimers(FALSE);
                    _progress := 350;
                END_IF;

                IF _progress = 350 THEN                                                                                     // TemplateTask_10steps_6 running: , add_the_detailed_description_of_the_current_action_1
                    IF _infoTimer.output THEN
                        TaskMessenger.Activate( UINT#550, eAxoMessageCategory#Warning);
                        Status.Error.Id :=      UINT#550;
                    END_IF;

                    IF TRUE THEN
                        THIS.CallTimers(FALSE);
                        _progress := 351;
                    END_IF;
                END_IF;

                IF _progress = 351 THEN                                                                                     // TemplateTask_10steps_6 running: , add_the_detailed_description_of_the_current_action_2
                    IF _infoTimer.output THEN
                        TaskMessenger.Activate( UINT#551, eAxoMessageCategory#Warning);
                        Status.Error.Id :=      UINT#551;
                    END_IF;

                    IF TRUE THEN
                        THIS.CallTimers(FALSE);
                        _progress := 352;
                    END_IF;
                END_IF;

                IF _progress = 352 THEN                                                                                     // TemplateTask_10steps_6 running: , add_the_detailed_description_of_the_current_action_3
                    IF _infoTimer.output THEN
                        TaskMessenger.Activate( UINT#552, eAxoMessageCategory#Warning);
                        Status.Error.Id :=      UINT#552;
                    END_IF;

                    IF TRUE THEN
                        THIS.CallTimers(FALSE);
                        _progress := 353;
                    END_IF;
                END_IF;

                IF _progress = 353 THEN                                                                                     // TemplateTask_10steps_6 running: , add_the_detailed_description_of_the_current_action_4
                    IF _infoTimer.output THEN
                        TaskMessenger.Activate( UINT#553, eAxoMessageCategory#Warning);
                        Status.Error.Id :=      UINT#553;
                    END_IF;

                    IF TRUE THEN
                        THIS.CallTimers(FALSE);
                        _progress := 354;
                    END_IF;
                END_IF;

                IF _progress = 354 THEN                                                                                     // TemplateTask_10steps_6 running: , add_the_detailed_description_of_the_current_action_5
                    IF _infoTimer.output THEN
                        TaskMessenger.Activate( UINT#554, eAxoMessageCategory#Warning);
                        Status.Error.Id :=      UINT#554;
                    END_IF;

                    IF TRUE THEN
                        THIS.CallTimers(FALSE);
                        _progress := 355;
                    END_IF;
                END_IF;

                IF _progress = 355 THEN                                                                                     // TemplateTask_10steps_6 running: , add_the_detailed_description_of_the_current_action_6
                    IF _infoTimer.output THEN
                        TaskMessenger.Activate( UINT#555, eAxoMessageCategory#Warning);
                        Status.Error.Id :=      UINT#555;
                    END_IF;

                    IF TRUE THEN
                        THIS.CallTimers(FALSE);
                        _progress := 356;
                    END_IF;
                END_IF;

                IF _progress = 356 THEN                                                                                     // TemplateTask_10steps_6 running: , add_the_detailed_description_of_the_current_action_7
                    IF _infoTimer.output THEN
                        TaskMessenger.Activate( UINT#556, eAxoMessageCategory#Warning);
                        Status.Error.Id :=      UINT#556;
                    END_IF;

                    IF TRUE THEN
                        THIS.CallTimers(FALSE);
                        _progress := 357;
                    END_IF;
                END_IF;

                IF _progress = 357 THEN                                                                                     // TemplateTask_10steps_6 running: , add_the_detailed_description_of_the_current_action_8
                    IF _infoTimer.output THEN
                        TaskMessenger.Activate( UINT#557, eAxoMessageCategory#Warning);
                        Status.Error.Id :=      UINT#557;
                    END_IF;

                    IF TRUE THEN
                        THIS.CallTimers(FALSE);
                        _progress := 358;
                    END_IF;
                END_IF;

                IF _progress = 358 THEN                                                                                     // TemplateTask_10steps_6 running: , add_the_detailed_description_of_the_current_action_9
                    IF _infoTimer.output THEN
                        TaskMessenger.Activate( UINT#558, eAxoMessageCategory#Warning);
                        Status.Error.Id :=      UINT#558;
                    END_IF;

                    IF TRUE THEN
                        THIS.CallTimers(FALSE);
                        _progress := 359;
                    END_IF;
                END_IF;

                IF _progress = 359 THEN                                                                                     // TemplateTask_10steps_6 running: , add_the_detailed_description_of_the_current_action_10
                    TemplateTask_10steps_6.DoneWhen(TRUE);
                    _progress := 0;
                END_IF;

                THIS.CallTimers(TRUE);

                TemplateTask_10steps_6.ThrowWhen(_errorTimer.output);
                Status.Action.Id := TO_UINT(_progress);
                TemplateTask_10steps_6.ThrowWhen(TemplateTask_10steps_6.Duration >= Config.TaskTimeout AND Config.TaskTimeout > T#0s ,'TemplateTask_10steps_6 timeout.');
            END_IF;
            IF TemplateTask_10steps_6.DoneReached() THEN
                Status.Action.Id :=  UINT#151;
                Status.Error.Id :=  UINT#0;
            ELSIF TemplateTask_10steps_6.ErrorOccured() THEN
                Status.Action.Id :=  UINT#10050;
                Status.Error.Id  :=  UINT#10050;
            ELSIF TemplateTask_10steps_6.AbortTriggered()THEN
                Status.Action.Id :=  UINT#10051;
                Status.Error.Id  :=  UINT#10051;
            END_IF;
            Messenger.ActivateOnCondition(ULINT#10050,TemplateTask_10steps_6.HasError(), eAxoMessageCategory#Error);
            Messenger.ActivateOnCondition(ULINT#10051,TemplateTask_10steps_6.IsAborted(), eAxoMessageCategory#Error);
            Messenger.ActivateOnCondition(ULINT#152,TemplateTask_10steps_6.RestoreTriggered() , eAxoMessageCategory#Error);
            IF TemplateTask_10steps_6.RestoreTriggered() AND _progress >= 350 AND _progress <= 359  THEN
                Status.Action.Id :=  UINT#152;
                _progress := 0;
            END_IF;
            //**************************************************

            //*************TemplateTask_20steps_1***************
            TemplateTask_20steps_1.SetIsDisabled(FALSE);
            IF TemplateTask_20steps_1.StartTriggered() THEN
                Status.Action.Id :=  UINT#160;
            END_IF;
            Messenger.ActivateOnCondition(ULINT#160,TemplateTask_20steps_1.IsBusy(), eAxoMessageCategory#Info);
            Messenger.ActivateOnCondition(ULINT#161,TemplateTask_20steps_1.IsDone(), eAxoMessageCategory#Info);
            IF TemplateTask_20steps_1.Execute(THIS) THEN
                IF _progress = 0 THEN
                    Status.Error.Id := UINT#0;
                    TaskMessenger.Restore();
                    THIS.CallTimers(FALSE);
                    _progress := 360;
                END_IF;

                IF _progress = 360 THEN                                                                                     // TemplateTask_20steps_1 running: , add_the_detailed_description_of_the_current_action_1
                    IF _infoTimer.output THEN
                        TaskMessenger.Activate( UINT#560, eAxoMessageCategory#Warning);
                        Status.Error.Id :=      UINT#560;
                    END_IF;

                    IF TRUE THEN
                        THIS.CallTimers(FALSE);
                        _progress := 361;
                    END_IF;
                END_IF;

                IF _progress = 361 THEN                                                                                     // TemplateTask_20steps_1 running: , add_the_detailed_description_of_the_current_action_2
                    IF _infoTimer.output THEN
                        TaskMessenger.Activate( UINT#561, eAxoMessageCategory#Warning);
                        Status.Error.Id :=      UINT#561;
                    END_IF;

                    IF TRUE THEN
                        THIS.CallTimers(FALSE);
                        _progress := 362;
                    END_IF;
                END_IF;

                IF _progress = 362 THEN                                                                                     // TemplateTask_20steps_1 running: , add_the_detailed_description_of_the_current_action_3
                    IF _infoTimer.output THEN
                        TaskMessenger.Activate( UINT#562, eAxoMessageCategory#Warning);
                        Status.Error.Id :=      UINT#562;
                    END_IF;

                    IF TRUE THEN
                        THIS.CallTimers(FALSE);
                        _progress := 363;
                    END_IF;
                END_IF;

                IF _progress = 363 THEN                                                                                     // TemplateTask_20steps_1 running: , add_the_detailed_description_of_the_current_action_4
                    IF _infoTimer.output THEN
                        TaskMessenger.Activate( UINT#563, eAxoMessageCategory#Warning);
                        Status.Error.Id :=      UINT#563;
                    END_IF;

                    IF TRUE THEN
                        THIS.CallTimers(FALSE);
                        _progress := 364;
                    END_IF;
                END_IF;

                IF _progress = 364 THEN                                                                                     // TemplateTask_20steps_1 running: , add_the_detailed_description_of_the_current_action_5
                    IF _infoTimer.output THEN
                        TaskMessenger.Activate( UINT#564, eAxoMessageCategory#Warning);
                        Status.Error.Id :=      UINT#564;
                    END_IF;

                    IF TRUE THEN
                        THIS.CallTimers(FALSE);
                        _progress := 365;
                    END_IF;
                END_IF;

                IF _progress = 365 THEN                                                                                     // TemplateTask_20steps_1 running: , add_the_detailed_description_of_the_current_action_6
                    IF _infoTimer.output THEN
                        TaskMessenger.Activate( UINT#565, eAxoMessageCategory#Warning);
                        Status.Error.Id :=      UINT#565;
                    END_IF;

                    IF TRUE THEN
                        THIS.CallTimers(FALSE);
                        _progress := 366;
                    END_IF;
                END_IF;

                IF _progress = 366 THEN                                                                                     // TemplateTask_20steps_1 running: , add_the_detailed_description_of_the_current_action_7
                    IF _infoTimer.output THEN
                        TaskMessenger.Activate( UINT#566, eAxoMessageCategory#Warning);
                        Status.Error.Id :=      UINT#566;
                    END_IF;

                    IF TRUE THEN
                        THIS.CallTimers(FALSE);
                        _progress := 367;
                    END_IF;
                END_IF;

                IF _progress = 367 THEN                                                                                     // TemplateTask_20steps_1 running: , add_the_detailed_description_of_the_current_action_8
                    IF _infoTimer.output THEN
                        TaskMessenger.Activate( UINT#567, eAxoMessageCategory#Warning);
                        Status.Error.Id :=      UINT#567;
                    END_IF;

                    IF TRUE THEN
                        THIS.CallTimers(FALSE);
                        _progress := 368;
                    END_IF;
                END_IF;

                IF _progress = 368 THEN                                                                                     // TemplateTask_20steps_1 running: , add_the_detailed_description_of_the_current_action_9
                    IF _infoTimer.output THEN
                        TaskMessenger.Activate( UINT#568, eAxoMessageCategory#Warning);
                        Status.Error.Id :=      UINT#568;
                    END_IF;

                    IF TRUE THEN
                        THIS.CallTimers(FALSE);
                        _progress := 369;
                    END_IF;
                END_IF;

                IF _progress = 369 THEN                                                                                     // TemplateTask_20steps_1 running: , add_the_detailed_description_of_the_current_action_10
                    IF _infoTimer.output THEN
                        TaskMessenger.Activate( UINT#569, eAxoMessageCategory#Warning);
                        Status.Error.Id :=      UINT#569;
                    END_IF;

                    IF TRUE THEN
                        THIS.CallTimers(FALSE);
                        _progress := 370;
                    END_IF;
                END_IF;

                IF _progress = 370 THEN                                                                                     // TemplateTask_20steps_1 running: , add_the_detailed_description_of_the_current_action_11
                    IF _infoTimer.output THEN
                        TaskMessenger.Activate( UINT#570, eAxoMessageCategory#Warning);
                        Status.Error.Id :=      UINT#570;
                    END_IF;

                    IF TRUE THEN
                        THIS.CallTimers(FALSE);
                        _progress := 371;
                    END_IF;
                END_IF;

                IF _progress = 371 THEN                                                                                     // TemplateTask_20steps_1 running: , add_the_detailed_description_of_the_current_action_12
                    IF _infoTimer.output THEN
                        TaskMessenger.Activate( UINT#571, eAxoMessageCategory#Warning);
                        Status.Error.Id :=      UINT#571;
                    END_IF;

                    IF TRUE THEN
                        THIS.CallTimers(FALSE);
                        _progress := 372;
                    END_IF;
                END_IF;

                IF _progress = 372 THEN                                                                                     // TemplateTask_20steps_1 running: , add_the_detailed_description_of_the_current_action_13
                    IF _infoTimer.output THEN
                        TaskMessenger.Activate( UINT#572, eAxoMessageCategory#Warning);
                        Status.Error.Id :=      UINT#572;
                    END_IF;

                    IF TRUE THEN
                        THIS.CallTimers(FALSE);
                        _progress := 373;
                    END_IF;
                END_IF;

                IF _progress = 373 THEN                                                                                     // TemplateTask_20steps_1 running: , add_the_detailed_description_of_the_current_action_14
                    IF _infoTimer.output THEN
                        TaskMessenger.Activate( UINT#573, eAxoMessageCategory#Warning);
                        Status.Error.Id :=      UINT#573;
                    END_IF;

                    IF TRUE THEN
                        THIS.CallTimers(FALSE);
                        _progress := 374;
                    END_IF;
                END_IF;

                IF _progress = 374 THEN                                                                                     // TemplateTask_20steps_1 running: , add_the_detailed_description_of_the_current_action_15
                    IF _infoTimer.output THEN
                        TaskMessenger.Activate( UINT#574, eAxoMessageCategory#Warning);
                        Status.Error.Id :=      UINT#574;
                    END_IF;

                    IF TRUE THEN
                        THIS.CallTimers(FALSE);
                        _progress := 375;
                    END_IF;
                END_IF;

                IF _progress = 375 THEN                                                                                     // TemplateTask_20steps_1 running: , add_the_detailed_description_of_the_current_action_16
                    IF _infoTimer.output THEN
                        TaskMessenger.Activate( UINT#575, eAxoMessageCategory#Warning);
                        Status.Error.Id :=      UINT#575;
                    END_IF;

                    IF TRUE THEN
                        THIS.CallTimers(FALSE);
                        _progress := 376;
                    END_IF;
                END_IF;

                IF _progress = 376 THEN                                                                                     // TemplateTask_20steps_1 running: , add_the_detailed_description_of_the_current_action_17
                    IF _infoTimer.output THEN
                        TaskMessenger.Activate( UINT#576, eAxoMessageCategory#Warning);
                        Status.Error.Id :=      UINT#576;
                    END_IF;

                    IF TRUE THEN
                        THIS.CallTimers(FALSE);
                        _progress := 377;
                    END_IF;
                END_IF;

                IF _progress = 377 THEN                                                                                     // TemplateTask_20steps_1 running: , add_the_detailed_description_of_the_current_action_18
                    IF _infoTimer.output THEN
                        TaskMessenger.Activate( UINT#577, eAxoMessageCategory#Warning);
                        Status.Error.Id :=      UINT#577;
                    END_IF;

                    IF TRUE THEN
                        THIS.CallTimers(FALSE);
                        _progress := 378;
                    END_IF;
                END_IF;

                IF _progress = 378 THEN                                                                                     // TemplateTask_20steps_1 running: , add_the_detailed_description_of_the_current_action_19
                    IF _infoTimer.output THEN
                        TaskMessenger.Activate( UINT#578, eAxoMessageCategory#Warning);
                        Status.Error.Id :=      UINT#578;
                    END_IF;

                    IF TRUE THEN
                        THIS.CallTimers(FALSE);
                        _progress := 379;
                    END_IF;
                END_IF;

                IF _progress = 379 THEN                                                                                     // TemplateTask_20steps_1 running: , add_the_detailed_description_of_the_current_action_20
                    TemplateTask_20steps_1.DoneWhen(TRUE);
                    _progress := 0;
                END_IF;

                THIS.CallTimers(TRUE);

                TemplateTask_20steps_1.ThrowWhen(_errorTimer.output);
                Status.Action.Id := TO_UINT(_progress);
                TemplateTask_20steps_1.ThrowWhen(TemplateTask_20steps_1.Duration >= Config.TaskTimeout AND Config.TaskTimeout > T#0s ,'TemplateTask_20steps_1 timeout.');
            END_IF;
            IF TemplateTask_20steps_1.DoneReached() THEN
                Status.Action.Id :=  UINT#161;
                Status.Error.Id :=  UINT#0;
            ELSIF TemplateTask_20steps_1.ErrorOccured() THEN
                Status.Action.Id :=  UINT#10060;
                Status.Error.Id  :=  UINT#10060;
            ELSIF TemplateTask_20steps_1.AbortTriggered()THEN
                Status.Action.Id :=  UINT#10061;
                Status.Error.Id  :=  UINT#10061;
            END_IF;
            Messenger.ActivateOnCondition(ULINT#10060,TemplateTask_20steps_1.HasError(), eAxoMessageCategory#Error);
            Messenger.ActivateOnCondition(ULINT#10061,TemplateTask_20steps_1.IsAborted(), eAxoMessageCategory#Error);
            Messenger.ActivateOnCondition(ULINT#162,TemplateTask_20steps_1.RestoreTriggered() , eAxoMessageCategory#Error);
            IF TemplateTask_20steps_1.RestoreTriggered() AND _progress >= 360 AND _progress <= 379  THEN
                Status.Action.Id :=  UINT#162;
                _progress := 0;
            END_IF;
            //**************************************************

            //*************TemplateTask_20steps_2***************
            TemplateTask_20steps_2.SetIsDisabled(FALSE);
            IF TemplateTask_20steps_2.StartTriggered() THEN
                Status.Action.Id :=  UINT#180;
            END_IF;
            Messenger.ActivateOnCondition(ULINT#180,TemplateTask_20steps_2.IsBusy(), eAxoMessageCategory#Info);
            Messenger.ActivateOnCondition(ULINT#181,TemplateTask_20steps_2.IsDone(), eAxoMessageCategory#Info);
            IF TemplateTask_20steps_2.Execute(THIS) THEN
                IF _progress = 0 THEN
                    Status.Error.Id := UINT#0;
                    TaskMessenger.Restore();
                    THIS.CallTimers(FALSE);
                    _progress := 380;
                END_IF;

                IF _progress = 380 THEN                                                                                     // TemplateTask_20steps_2 running: , add_the_detailed_description_of_the_current_action_1
                    IF _infoTimer.output THEN
                        TaskMessenger.Activate( UINT#580, eAxoMessageCategory#Warning);
                        Status.Error.Id :=      UINT#580;
                    END_IF;

                    IF TRUE THEN
                        THIS.CallTimers(FALSE);
                        _progress := 381;
                    END_IF;
                END_IF;

                IF _progress = 381 THEN                                                                                     // TemplateTask_20steps_2 running: , add_the_detailed_description_of_the_current_action_2
                    IF _infoTimer.output THEN
                        TaskMessenger.Activate( UINT#581, eAxoMessageCategory#Warning);
                        Status.Error.Id :=      UINT#581;
                    END_IF;

                    IF TRUE THEN
                        THIS.CallTimers(FALSE);
                        _progress := 382;
                    END_IF;
                END_IF;

                IF _progress = 382 THEN                                                                                     // TemplateTask_20steps_2 running: , add_the_detailed_description_of_the_current_action_3
                    IF _infoTimer.output THEN
                        TaskMessenger.Activate( UINT#582, eAxoMessageCategory#Warning);
                        Status.Error.Id :=      UINT#582;
                    END_IF;

                    IF TRUE THEN
                        THIS.CallTimers(FALSE);
                        _progress := 383;
                    END_IF;
                END_IF;

                IF _progress = 383 THEN                                                                                     // TemplateTask_20steps_2 running: , add_the_detailed_description_of_the_current_action_4
                    IF _infoTimer.output THEN
                        TaskMessenger.Activate( UINT#583, eAxoMessageCategory#Warning);
                        Status.Error.Id :=      UINT#583;
                    END_IF;

                    IF TRUE THEN
                        THIS.CallTimers(FALSE);
                        _progress := 384;
                    END_IF;
                END_IF;

                IF _progress = 384 THEN                                                                                     // TemplateTask_20steps_2 running: , add_the_detailed_description_of_the_current_action_5
                    IF _infoTimer.output THEN
                        TaskMessenger.Activate( UINT#584, eAxoMessageCategory#Warning);
                        Status.Error.Id :=      UINT#584;
                    END_IF;

                    IF TRUE THEN
                        THIS.CallTimers(FALSE);
                        _progress := 385;
                    END_IF;
                END_IF;

                IF _progress = 385 THEN                                                                                     // TemplateTask_20steps_2 running: , add_the_detailed_description_of_the_current_action_6
                    IF _infoTimer.output THEN
                        TaskMessenger.Activate( UINT#585, eAxoMessageCategory#Warning);
                        Status.Error.Id :=      UINT#585;
                    END_IF;

                    IF TRUE THEN
                        THIS.CallTimers(FALSE);
                        _progress := 386;
                    END_IF;
                END_IF;

                IF _progress = 386 THEN                                                                                     // TemplateTask_20steps_2 running: , add_the_detailed_description_of_the_current_action_7
                    IF _infoTimer.output THEN
                        TaskMessenger.Activate( UINT#586, eAxoMessageCategory#Warning);
                        Status.Error.Id :=      UINT#586;
                    END_IF;
